{attribute 'linkalways'} 
{attribute 'no_explicit_call' := 'This FB is a CLASS and must be accessed using methods or properties'}
{attribute 'enable_dynamic_creation'}
FUNCTION_BLOCK FINAL GE_UINT EXTENDS Node
VAR
	in1 : _UINT(0);
	in2 : _UINT(0);
	out : _BOOL(FALSE);
END_VAR

METHOD PUBLIC Clone : I_Node
VAR
	pNode : POINTER TO GE_UINT;
END_VAR
pNode := __NEW(GE_UINT);
Clone := pNode^;
END_METHOD

METHOD FB_init : BOOL
VAR_INPUT
	bInitRetains : BOOL; // if TRUE, the retain variables are initialized (warm start / cold start)
	bInCopyCode : BOOL;  // if TRUE, the instance afterwards gets moved into the copy code (online change)
END_VAR
AddInput('in1',THIS^.in1);
AddInput('in2',THIS^.in2);
AddOutput('out', THIS^.out);
END_METHOD

METHOD PROTECTED OnExecute
VAR
END_VAR
out.Value := in1.Value >= in2.Value;
END_METHOD

END_FUNCTION_BLOCK

(* stored: Version 1.1.0.1, ProductVersion 3.1.4024.15
   POU GE_UINT: Id {2d211557-3f4c-4f7c-88a8-26cef6e77dd5}, SpecialFunc None
   Folder Constructor: Id {99efb80d-9fa5-4f97-a402-3170b44f9210}
   Method Clone: Id {83798e7c-fd30-40d8-b148-2747cfd6b61b}
   Method FB_init: Id {ea00b7da-e6fe-4790-9b82-68f01cafe57d}
   Method OnExecute: Id {a1dc37e0-31ac-45d4-851e-944d9cc1d02d} *)
